PROGRAM PRG_10_Persistent
VAR
	fb_UPS: FB_S_UPS_CX51x0;
END_VAR

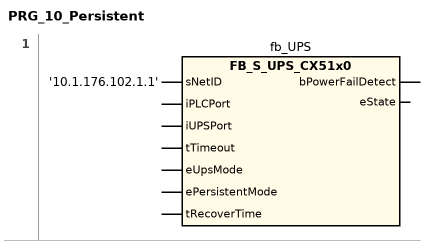
// NETWORK 1
fb_UPS(sNetID := '10.1.176.102.1.1'); // FB_S_UPS_CX51x0

END_PROGRAM

(* stored: Version 1.1.0.1, ProductVersion 3.1.4024.12
   POU PRG_10_Persistent: Id {f3a92364-9450-458d-9c21-d9eea605a570}, SpecialFunc None *)
